{attribute 'qualified_only'}
{attribute 'strict'}
TYPE E_StopCodes :
(
	NoStop := 0,
	SystemStop := 1,
	MotorOL := 2,
	VFD_Fault := 3,
	ProductJam := 4,
	MotorRunTO := 5,
	VFDRunTO := 6,
	LowAir := 7,
	MergeJam := 8,
	SlackBeltFault := 9,
	EncoderFault := 10,
	TransferTO := 11,
	TransferLP := 12,
	ActuatorTO := 13,
	SprialTorque := 14,
	DisconnectState := 15,
	ReleaseFault := 16,
	PanelIOFLT := 17,
	FieldIOFLT := 18,
	UnderHeightFLT := 19,
	OverHeightFLT := 20,
	Taper :=21,
	DeviceNoInAuto := 22
) UINT;
END_TYPE

(* stored: Version 1.1.0.1, ProductVersion 3.1.4024.4
   EnumerationTextList E_StopCodes: Id {74aa730f-5a7b-4a80-b7af-f961e7835c4b} *)
